{library PUBLIC}
(* Use this function block to initiate, maintain and end a session. The session is queued
    when En=TRUE, when a session is possible Established is set to True. If En becomes FALSE and the a session is queued (waiting) the 
    session is aborted. However, if a session is established ongoing transmistion is not aborted.  To abort an ongoing transmission set En to FALSE 
   and disable the he Communicator block (En=FALSE) at the same time.
*)
FUNCTION_BLOCK SessionInit
VAR_INPUT
	En:					BOOL:=FALSE;			(* Set to true to Initiate and maintain a session and to end a session or abort set to low *)
END_VAR
VAR_OUTPUT
	Done:				BOOL:=FALSE;			(* Set to true when En is true and a session is established, set to false when En is false *)
	Established:		BOOL:=FALSE;			(* True if a session is established *)
	SessionID:		INT:=-1;					(* A  session ID number or -1 if no active session *)
END_VAR
VAR_IN_OUT
	Data: 				CommunicationData;		(* Common data structure to connect this function block to a specific Communicator block *)
END_VAR
VAR
	Sequence: 		INT := 0;
END_VAR

IF En THEN
	CASE Sequence OF
		0: (* Wait until possible to get a session *)
			IF NOT Data._Session._Locked AND Data._Status=DATAGRAM_SEQUENCE.DATAGRAM_SEQUENCE_NOP AND Data._DataExecute=Data._DataCounter THEN
				Data._Session._Locked:=TRUE;
				Data._Session._SessionID:=Data._Session._SessionID+1;
				Data._Session._SessionCounter:=0;
				Data._Session._SessionBussy:=FALSE;
				Data._DataExecute:=0;
				Data._DataCounter:=0;

				SessionID:=Data._Session._SessionID;
				Established:=TRUE;
				Done:=TRUE;
				Sequence:=1;
			END_IF;

		1:
			(* Some one else has closed the session *)
			IF NOT Data._Session._Locked OR SessionID<>Data._Session._SessionID THEN
				Established:=FALSE;
				SessionID:=-1;
			END_IF;
	END_CASE;
ELSE
	Sequence:=0;
	Done:=FALSE;
 	IF Established THEN
		Data._Session._Locked:=FALSE;
		Established:=FALSE;
		SessionID:=-1;
	END_IF;
END_IF;

END_FUNCTION_BLOCK

(* stored: Version 1.1.0.1, ProductVersion 3.1.4024.2
   POU SessionInit: Id {fef3df90-16a8-45ce-aa52-9322fb8ed0c3}, SpecialFunc None *)
